{attribute 'qualified_only'}
{attribute 'strict'}
TYPE E_STATES_BOHRKOPF :
(
	initializing := 0,
	stopped,
	stopping,
	ready,
	going_down,
	going_up
);
END_TYPE

(* stored: Version 1.1.0.1, ProductVersion 3.1.4024.3
   DUT E_STATES_BOHRKOPF: Id {de10afe8-dac8-437b-ba8f-1b6821160c33} *)
